KUKA KRL data list: G1_test.dat

&ACCESS RVO1
&COMMENT Modul (src/dat) with INI line and PTP HOME at start and end of Program
DEFDAT G1_test PUBLIC
;FOLD EXTERNAL DECLARATIONS;%{PE}%MKUKATPBASIS,%CEXT,%VCOMMON,%P
;FOLD BASISTECH EXT;%{PE}%MKUKATPBASIS,%CEXT,%VEXT,%P
EXT  BAS (BAS_COMMAND  :IN,REAL  :IN )
DECL INT SUCCESS
;ENDFOLD (BASISTECH EXT)
;FOLD USER EXT;%{E}%MKUKATPUSER,%CEXT,%VEXT,%P
;Make here your modifications

;ENDFOLD (USER EXT)
;ENDFOLD (EXTERNAL DECLERATIONS)
DECL E6POS XP1={X 0,Y 0,Z 0,A 0,B 0,C 0,S 0,T 0,E1 0,E2 0,E3 0,E4 0,E5 0,E6 0}
DECL FDAT FP1={TOOL_NO 1,BASE_NO 1,IPO_FRAME #BASE,POINT2[] " ",TQ_STATE FALSE}
DECL E6POS XP2={X 0,Y 0,Z 0,A 0,B 0,C 0,S 0,T 0,E1 0,E2 0,E3 0,E4 0,E5 0,E6 0}
DECL FDAT FP2={TOOL_NO 1,BASE_NO 1,IPO_FRAME #BASE,POINT2[] " ",TQ_STATE FALSE}
DECL PDAT PPDAT21={VEL 100,ACC 100,APO_DIST 100,APO_MODE #CPTP,GEAR_JERK 50}
DECL E6POS XP3={X 0,Y 0,Z 0,A 0,B 0,C 0,S 0,T 0,E1 0,E2 0,E3 0,E4 0,E5 0,E6 0}
DECL FDAT FP3={TOOL_NO 1,BASE_NO 1,IPO_FRAME #BASE,POINT2[] " ",TQ_STATE FALSE}
DECL PDAT PPDAT22={VEL 100,ACC 100,APO_DIST 100,APO_MODE #CPTP,GEAR_JERK 50}
DECL E6POS XP4={X 0,Y 0,Z 0,A 0,B 0,C 0,S 0,T 0,E1 0,E2 0,E3 0,E4 0,E5 0,E6 0}
DECL FDAT FP4={TOOL_NO 1,BASE_NO 1,IPO_FRAME #BASE,POINT2[] " ",TQ_STATE FALSE}
DECL PDAT PPDAT23={VEL 100,ACC 100,APO_DIST 100,APO_MODE #CPTP,GEAR_JERK 50}
DECL E6POS Xmusic[0].x={X 0,Y 0,Z 0,A 0,B 0,C 0,S 0,T 0,E1 0,E2 0,E3 0,E4 0,E5 0,E6 0}
DECL FDAT Fmusic[0].x={TOOL_NO 0,BASE_NO 0,IPO_FRAME #BASE,POINT2[] " ",TQ_STATE FALSE}
DECL PDAT PPDAT0={VEL 100,ACC 100,APO_DIST 100,APO_MODE #CPTP,GEAR_JERK 50}
DECL E6POS Xmusic[0].x={X 0,Y 0,Z 0,A 0,B 0,C 0,S 0,T 0,E1 0,E2 0,E3 0,E4 0,E5 0,E6 0}
DECL FDAT Fmusic[0].x={TOOL_NO 0,BASE_NO 0,IPO_FRAME #BASE,POINT2[] " ",TQ_STATE FALSE}
DECL E6POS Xmusic[0].x={X 0,Y 0,Z 0,A 0,B 0,C 0,S 0,T 0,E1 0,E2 0,E3 0,E4 0,E5 0,E6 0}
DECL FDAT Fmusic[0].x={TOOL_NO 1,BASE_NO 1,IPO_FRAME #BASE,POINT2[] " ",TQ_STATE FALSE}
DECL E6POS Xmusic[0].x+10={X 0,Y 0,Z 0,A 0,B 0,C 0,S 0,T 0,E1 0,E2 0,E3 0,E4 0,E5 0,E6 0}
DECL FDAT Fmusic[0].x+10={TOOL_NO 1,BASE_NO 1,IPO_FRAME #BASE,POINT2[] " ",TQ_STATE FALSE}
DECL E6POS Xmusic[0].x+10={X 0,Y 0,Z 0,A 0,B 0,C 0,S 0,T 0,E1 0,E2 0,E3 0,E4 0,E5 0,E6 0}
DECL FDAT Fmusic[0].x+10={TOOL_NO 1,BASE_NO 1,IPO_FRAME #BASE,POINT2[] " ",TQ_STATE FALSE}
DECL E6POS Xmusic[0].x={X 0,Y 0,Z 0,A 0,B 0,C 0,S 0,T 0,E1 0,E2 0,E3 0,E4 0,E5 0,E6 0}
DECL FDAT Fmusic[0].x={TOOL_NO 1,BASE_NO 1,IPO_FRAME #BASE,POINT2[] " ",TQ_STATE FALSE}
DECL E6POS XP1[0]={X 0,Y 0,Z 0,A 0,B 0,C 0,S 0,T 0,E1 0,E2 0,E3 0,E4 0,E5 0,E6 0}
DECL FDAT FP1[0]={TOOL_NO 1,BASE_NO 1,IPO_FRAME #BASE,POINT2[] " ",TQ_STATE FALSE}
ENDDAT
